TYPE E_CX_DeviceState_1 : (
	E_CX_DEVICE_IDLE,
	E_CX_DEVICE_ID,
	E_CX_DEVICE_TYPE,
	E_CX_DEVICE_BUILDLINES,
	E_CX_DEVICE_WRITELINE1,
	E_CX_DEVICE_WRITELINE2,
	E_CX_DEVICE_DONE,
	E_CX_DEVICE_ERROR,
	E_CX_DEVICE_CX1,
	E_CX_DEVICE_CX2
);
END_TYPE

(* stored: Version 1.1.0.1
   DUT E_CX_DeviceState_1: Id {6601a748-4cdd-4e82-987d-3f07d2b835a4} *)
